# EPICS substitutions: db/Beckhoff_1XXX/ecmcCU1561.substitutions
file "empty.template"{
  pattern {}
}
